ABB RobotStudio station: simulación_1_cilindro.rsstn

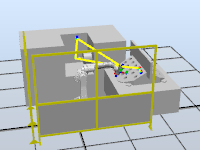
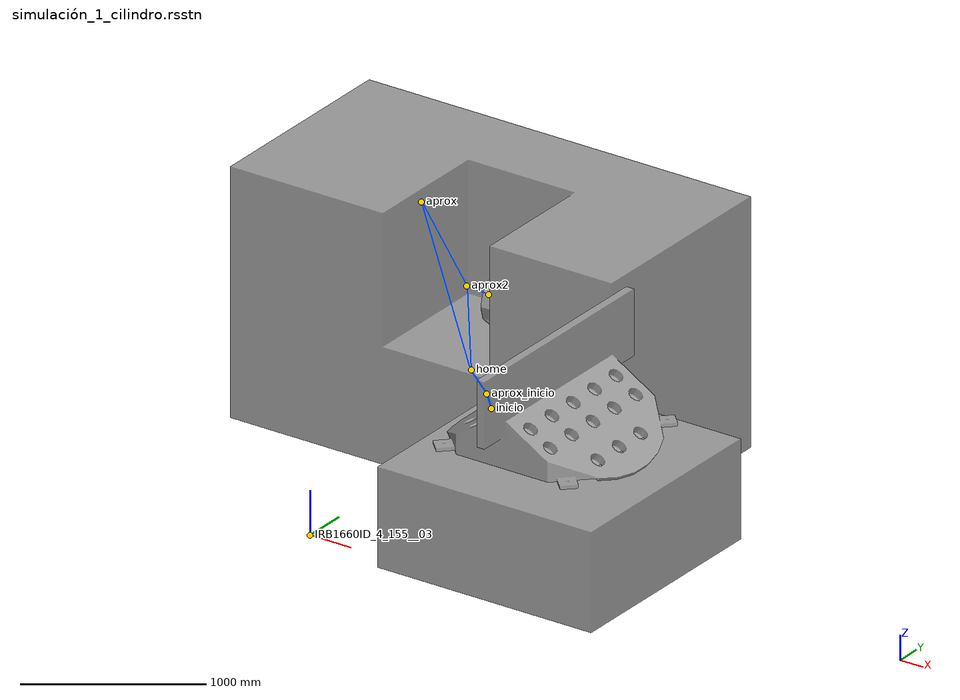
[picture v1: parts stored in the station drawn from their meshes, with robot base, taught points and paths (robot models come from the ABB library and are not in the file)]
Station Station (saved by RobotStudio 21.4.9700.0)
Controller Controller1
  mechanical unit ROB_1: IRB1660ID_4_155__03, 6 joints, base frame (0, 0, 0) mm
Layout (positions relative to the parent item):
  - Pinza_1 [mechanism, from Efectores_finales - Copy\PinzaF_1.rslib] at (944.87, 0, 1229) mm, rotated rx -180 ry 60 rz -180 deg; joint values [0, 0] (rad or m)
  - Pinza_2 [mechanism, from Efectores_finales - Copy\PinzaF_2.rslib] at (944.87, 0, 1229) mm, rotated rx -180 ry 60 rz -180 deg; joint values [0, 0] (rad or m)
  - IRB1660ID_4_155__03 [mechanism, from Robots\IRB1660ID_4_155__03.rslib] at (0, 0, 0) mm; joint values [0, 0, 0, 0, 0.5236, 0] (rad or m)
  - Attacher [smart component, from Components\Attacher.rslib]
      properties: Parent=Pinza_1; Flange=0; Child=Cilindros_2; Mount=false; Offset=[0 0 0]; Orientation=[0 0 0]
  - CollisionSensor [smart component, from Components\CollisionSensor.rslib]
      properties: Object1=Pinza_1; Object2=Cilindros_2; NearMiss=0.001; Part1=(none); Part2=(none); CollisionType=0
  - CollisionSensor_2 [smart component, from Components\CollisionSensor.rslib]
      properties: Object1=Cilindros_2; Object2=Cilindros_3; NearMiss=0.0005; Part1=Cilindros_2; Part2=Cilindros_3; CollisionType=2
  - Detacher [smart component, from Components\Detacher.rslib]
      properties: Child=Cilindros_2; KeepPosition=true
  - Positioner [smart component, from Components\Positioner.rslib]
      properties: Object=(none); Position=[0 0 0]; Orientation=[0 0 0]; Reference=Global; ReferenceObject=(none)
  - Cilindros_2 [part] at (439.73, 1172.03, 1064.12) mm, rotated rx -117.01 ry -81.37 rz -62.71 deg, size 80 x 79.4 x 100 mm
  - Cilindros_3 [part] at (440.58, 1171.74, 1067.85) mm, rotated rx 0 ry -90 rz 0 deg, size 80 x 79.4 x 100 mm
  - Conjunto_para_piezas_huecos [part] at (976.83, 1711.44, 737.97) mm, rotated rx 90 ry 0 rz 0 deg, size 1400 x 1300 x 1400 mm
  - Torno [part] at (1400.58, 2121.74, 1567.85) mm, rotated rx 0 ry 0 rz 180 deg, size 2500 x 1300 x 1500 mm
  - Fence_740 [graphiccomponentgroup, from Equipment\Fence_740.rslib] at (-1013.32, -651.89, 5.82) mm
    - Body 1 [part, from Equipment\Fence_740.rslib]
    - Body 2 [part, from Equipment\Fence_740.rslib]
  - Fence_2500 [graphiccomponentgroup, from Equipment\Fence_2500.rslib] at (-892.95, -659.41, 0) mm, rotated rx 0 ry 0 rz -90 deg
    - Body 1 [part, from Equipment\Fence_2500.rslib]
    - Body 2 [part, from Equipment\Fence_2500.rslib]
  - Fence_740_2 [graphiccomponentgroup, from Equipment\Fence_740.rslib] at (-1000.12, 93.34, 0) mm
    - Body 1 [part, from Equipment\Fence_740.rslib]
    - Body 2 [part, from Equipment\Fence_740.rslib]
Attachment: Pinza_1 is attached to IRB1660ID_4_155__03 / Link6
Attachment: Pinza_2 is attached to IRB1660ID_4_155__03 / Link6
Station logic (signal -> signal, property => property):
  CollisionSensor.SensorOut -> Attacher.Execute
  CollisionSensor_2.SensorOut -> Detacher.Execute
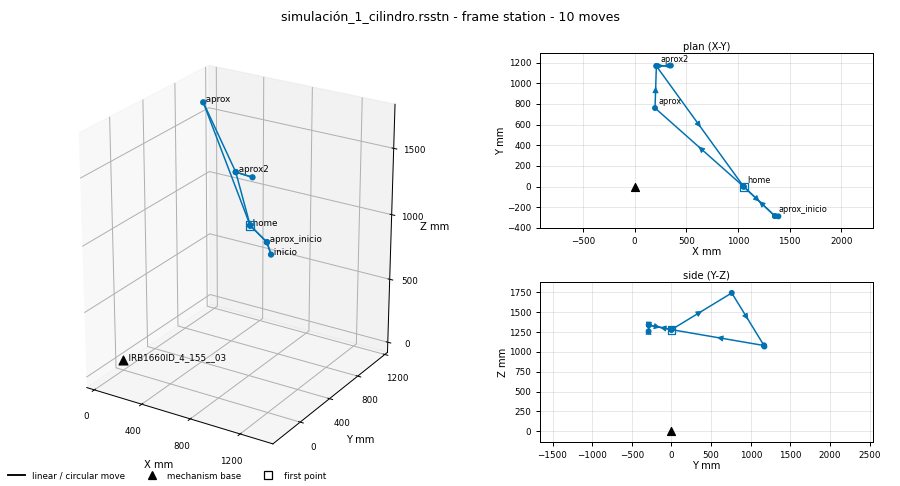
[picture p0: tool path of simulación_1_cilindro.rsstn in frame station, 10 of 10 moves have a stored position in this frame; points joined in program order, loops and branches not executed]
Targets, tools, work objects and paths stored in the station, written as RAPID:
! task T_ROB1
MODULE CalibData
  PERS tooldata Pinza_1:=[TRUE,[[-100,0,70],[0.707106781,0,-0.707106781,0]],[1,[0,0,1],[1,0,0,0],0,0,0]];
  PERS tooldata Vara:=[TRUE,[[0,0,250],[0.707106781,0,0,0.707106781]],[1,[0,0,1],[1,0,0,0],0,0,0]];
  PERS tooldata Soplador:=[TRUE,[[0,-70,70],[0.5,0.5,-0.5,0.5]],[1,[0,0,1],[1,0,0,0],0,0,0]];
  PERS tooldata Pinza_2_1:=[TRUE,[[100,0,70],[0.707106781,0,0.707106781,0]],[1,[0,0,2],[1,0,0,0],0,0,0]];
  TASK PERS wobjdata Workobject_1:=[FALSE,TRUE,"",[[0,0,0],[1,0,0,0]],[[0,0,0],[1,0,0,0]]];
ENDMODULE

! task T_ROB1
MODULE Module1
  CONST robtarget inicio:=[[1392.200443648,-288.557,1259.602883858],[0,0.970295726,0,0.241921895],[0,0,0,0],[9E+09,9E+09,9E+09,9E+09,9E+09,9E+09]];
  CONST robtarget fin:=[[350.583,1171.739,1067.848],[0.707106781,0,0.707106781,0],[0,0,0,0],[9E+09,9E+09,9E+09,9E+09,9E+09,9E+09]];
  CONST robtarget home:=[[1055.495207776,0,1280.602540378],[0.965925826,0,0.258819045,0],[0,0,0,0],[9E+09,9E+09,9E+09,9E+09,9E+09,9E+09]];
  CONST robtarget aprox:=[[197.776925294,760.03861872,1743.411454959],[0.791008439,0.011521125,-0.014902831,0.611515183],[0,0,-1,0],[9E+09,9E+09,9E+09,9E+09,9E+09,9E+09]];
  CONST robtarget aprox2:=[[210.807412786,1166.825154663,1080.299278128],[0.528354623,0.464080073,0.534342598,0.468987278],[0,1,-1,0],[9E+09,9E+09,9E+09,9E+09,9E+09,9E+09]];
  CONST robtarget aprox_inicio:=[[1358.892893102,-286.119771001,1338.241912639],[0.004703554,0.965367081,0.001172734,0.260850341],[-1,1,0,0],[9E+09,9E+09,9E+09,9E+09,9E+09,9E+09]];
  PROC main()
  ENDPROC
  PROC Path_10()
    MoveL home,v200,z5,Pinza_1\WObj:=Workobject_1;
    MoveL aprox_inicio,v200,z5,Pinza_1\WObj:=Workobject_1;
    MoveL inicio,v200,z5,Pinza_1\WObj:=Workobject_1;
    MoveL aprox_inicio,v200,z5,Pinza_1\WObj:=Workobject_1;
    MoveL home,v200,z5,Pinza_1\WObj:=Workobject_1;
    MoveL aprox,v200,z5,Pinza_1\WObj:=Workobject_1;
    MoveL aprox2,v200,z5,Pinza_1\WObj:=Workobject_1;
    MoveL fin,v200,z5,Pinza_1\WObj:=Workobject_1;
    MoveL aprox2,v200,z5,Pinza_1\WObj:=Workobject_1;
    MoveL home,v200,z5,Pinza_1\WObj:=Workobject_1;
  ENDPROC
ENDMODULE

